INTERFACE I_MoverApplication

METHOD Cycle
END_METHOD

PROPERTY P_nMoverIndex : INT
GET
END_GET
SET
END_SET
END_PROPERTY

PROPERTY P_nTrackId : UDINT
GET
END_GET
SET
END_SET
END_PROPERTY

PROPERTY std : I_XPlanarMoverStandard
GET
END_GET
SET
END_SET
END_PROPERTY

END_INTERFACE

(* stored: Version 1.1.0.1
   Itf I_MoverApplication: Id {e063d166-58d5-4cf3-9667-4435b8f50264}
   Method Cycle: Id {c5bb2867-ba70-4404-bbd6-f781660c832f}
   Property P_nMoverIndex: Id {46de7149-b83d-49e9-bb46-60e703c03568}
   Get Get: Id {b4101762-c762-4e64-8fba-4724bf4e30c9}
   Set Set: Id {aeaf9d9c-09c3-4e1b-8325-683cc883439a}
   Property P_nTrackId: Id {5e00ac0b-4280-4c12-b31b-0450a5fedbf9}
   Get Get: Id {eb990daf-3754-48fc-bb24-a27d6937a44f}
   Set Set: Id {b4af4069-2855-49d6-83d9-8396e4a29bbe}
   Property std: Id {86ac2f04-4369-4764-9195-431b2d989a7e}
   Get Get: Id {d4957e6f-f43e-4a93-a11a-9872914a031d}
   Set Set: Id {f0c5a095-ab67-4be2-adb5-00d65355a95d} *)
